// TIA Portal V19 export
DATA_BLOCK "IPC_Com_Channel_LOG_MES"   // DB13
// stored: MemoryReserve 100
   VAR
      RECEIVE : Struct   // Ricezione singolo messaggio da MES
         ack : DInt;   // Acknowledge msg.ID to MES
         msg : "IPC_Msg_Generico";
      END_STRUCT;
      SEND : Struct   // Invio singolo messaggio a MES
         ack : DInt;   // Acknowledge msg.ID From MES
         msg : "IPC_Msg_Log_MES";
      END_STRUCT;
   END_VAR
BEGIN
END_DATA_BLOCK
